(* CoDeSys 2.3.9.37 project: Cap11_10.pro *)
(* Libraries: Standard.lib 4.10.05 12:14:46, IecSfc.lib 13.4.06 16:51:28 *)

(* Global variable list: Global_Variables *)
VAR_GLOBAL

      (*Entradas*)
      START:BOOL;
	A1:BOOL;
	B1:BOOL;
	A2:BOOL;
	B2:BOOL;

       (* Salidas *)
	MOTOR_IZ1:BOOL;
	MOTOR_DE1:BOOL;
       MOTOR_IZ2:BOOL;
	MOTOR_DE2:BOOL;

      (* Variables del simulador *)
	Vel:INT:=1;
	Vel2:INT:=1;
END_VAR

(* POU PLC_PRG, FBD *)
PROGRAM PLC_PRG
VAR

END_VAR
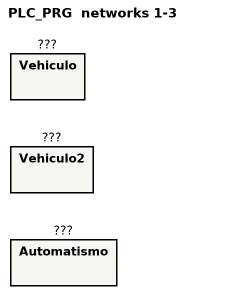
_FBD_ (* Function Block Diagram *)
NETWORK 1
	???:Vehiculo()
NETWORK 2
	???:Vehiculo2()
NETWORK 3
	???:Automatismo()
_END_FBD_
END_PROGRAM

(* POU Vehiculo, ST *)
PROGRAM Vehiculo
VAR
	PosX: INT;
END_VAR
A1:=FALSE;
B1:=FALSE;


IF MOTOR_DE1=TRUE THEN

     PosX:=PosX+Vel;

END_IF

IF MOTOR_IZ1=TRUE THEN

     PosX:=PosX-Vel;

END_IF


IF PosX<=0 THEN
   A1:=TRUE;
END_IF

IF PosX>=400 THEN
  B1:=TRUE;
END_IF
END_PROGRAM

(* POU Vehiculo2, ST *)
PROGRAM Vehiculo2
VAR
	PosX2: INT;
END_VAR
A2:=FALSE;
B2:=FALSE;


IF MOTOR_DE2=TRUE THEN

     PosX2:=PosX2+Vel2;

END_IF

IF MOTOR_IZ2=TRUE THEN

     PosX2:=PosX2-Vel2;

END_IF


IF PosX2<=0 THEN
   A2:=TRUE;
END_IF

IF PosX2>=400 THEN
  B2:=TRUE;
END_IF
END_PROGRAM

(* POU Automatismo, SFC *)
PROGRAM Automatismo
VAR
END_VAR
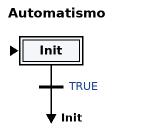
INITIAL_STEP Init:
END_STEP
TRANSITION FROM Init TO Init := TRUE;
END_TRANSITION
END_PROGRAM

(* Visualisation Vehiculo
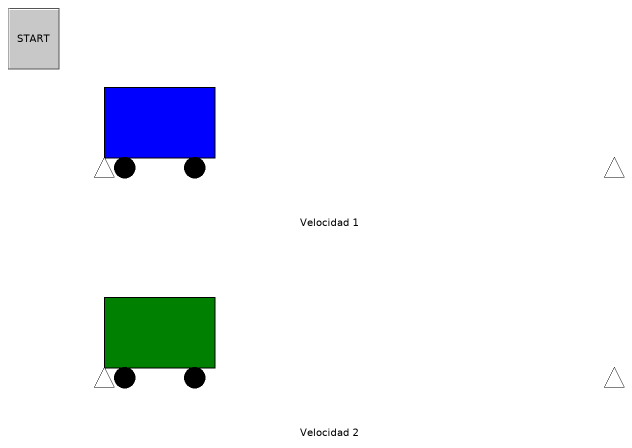
rectangle at (140,120)-(251,191): x offset Vehiculo.PosX
polygon at (130,190)-(150,210): alarm colour if .A1
polygon at (640,190)-(660,210): alarm colour if .B1
button at (44,41)-(95,102): text "START"; toggles START
rectangle at (140,330)-(251,401): x offset Vehiculo2.PosX2
polygon at (130,400)-(150,420): alarm colour if .A2
polygon at (640,400)-(660,420): alarm colour if .B2
ellipse at (150,190)-(171,211): x offset Vehiculo.PosX
ellipse at (220,190)-(241,211): x offset Vehiculo.PosX
ellipse at (150,400)-(171,421): x offset Vehiculo2.PosX2
ellipse at (220,400)-(241,421): x offset Vehiculo2.PosX2
rectangle at (310,240)-(421,271): text "Velocidad 1"
rectangle at (310,450)-(421,481): text "Velocidad 2"
2 elements of other kinds (tables, trends, ...) not read
*)
